GLOBALCONSTANTS AID_ON (* Output number object attribute ids *)
  (* Standard: 61499-1; Description: Copyright (c) 2023 HR Agrartechnik GmbH This program and the accompanying materials are made available under the terms of the Eclipse Public License 2.0 which is available at https://www.eclipse.org/legal/epl-2.0/ SPDX-License-Identifier: EPL-2.0 *)
  (* Version 1.0, 2026-06-20, Franz Höpfinger, HR Agrartechnik GmbH *)
  PACKAGE isobus::UT::Q::const::AID;
  VAR_GLOBAL CONSTANT
    WIDTH : USINT := USINT#1; (* 1: AID_ON_WIDTH - Width in pixels. *)
    HEIGHT : USINT := USINT#2; (* 2: AID_ON_HEIGHT - Height in pixels. *)
    BACKGROUND_COLOUR : USINT := USINT#3; (* 3: AID_ON_BACKGROUND_COLOUR - Background colour index. *)
    FONT_ATT : USINT := USINT#4; (* 4: AID_ON_FONT_ATT - Object ID of a Font Attributes object. *)
    OPTIONS : USINT := USINT#5; (* 5: AID_ON_OPTIONS - Options bitmask. *)
    VARIABLE_REF : USINT := USINT#6; (* 6: AID_ON_VARIABLE_REF - Object ID of a Number Variable object. *)
    OFFSET : USINT := USINT#7; (* 7: AID_ON_OFFSET - Offset to be applied to the value for display. *)
    SCALE : USINT := USINT#8; (* 8: AID_ON_SCALE - Scale to be applied to the value for display. *)
    NUMB_DECIMALS : USINT := USINT#9; (* 9: AID_ON_NUMB_DECIMALS - Number of decimals to display after the decimal point. *)
    FORMAT : USINT := USINT#10; (* 10: AID_ON_FORMAT - 0 = fixed format decimal (####.nn), 1 = exponential format. *)
    JUSTIFICATION : USINT := USINT#11; (* 11: AID_ON_JUSTIFICATION - Justification: Bits 0-1 (Horizontal: 0=Left, 1=Middle, 2=Right), Bits *)
    VALUE : USINT := USINT#12; (* 12: AID_ON_VALUE (read-only) - Current value before scaling. *)
  END_VAR
END_GLOBALCONSTANTS
